// TIA Portal V17 export
// export: Created 2022-02-03T14:45:13.9253235Z, ExportSetting WithDefaults, DisplayName Totally Integrated Automation Portal, DisplayVersion V17, DisplayName TIA Portal Openness, DisplayVersion V17, DisplayName TIA Portal Version Control Interface, DisplayVersion V17, DisplayName SINAMICS Startdrive Advanced, DisplayVersion V17, DisplayName SINAMICS Startdrive G130, G150, S120, S150, SINAMICS MV, S210, DisplayVersion V17, DisplayName SINAMICS Startdrive G110M, G120, G120C, G120D, G120P, G115D, DisplayVersion V17, DisplayName STEP 7 Professional, DisplayVersion V17, DisplayName STEP 7 Safety, DisplayVersion V17, DisplayName WinCC Advanced, DisplayVersion V17
ORGANIZATION_BLOCK "Pull or plug of modules"   // OB83, LAD, PullOrPlugOfModules
VERSION : 0.1
// stored: IsIECCheckEnabled false, SetENOAutomatically false
   VAR_INPUT
      LADDR : HW_IO;   // Hardware identifier
      Event_Class : Byte;   // 16#38/39: module inserted, removed
      Fault_ID : Byte;   // Fault identifier
   END_VAR
   VAR_TEMP
      tempAddress : GEOADDR;
      temp_RetVal : Word;
   END_VAR
   VAR_TEMP   // added for the SCL form of the ladder/FBD networks
      _w1 : Bool;
   END_VAR
BEGIN

REGION Network 1
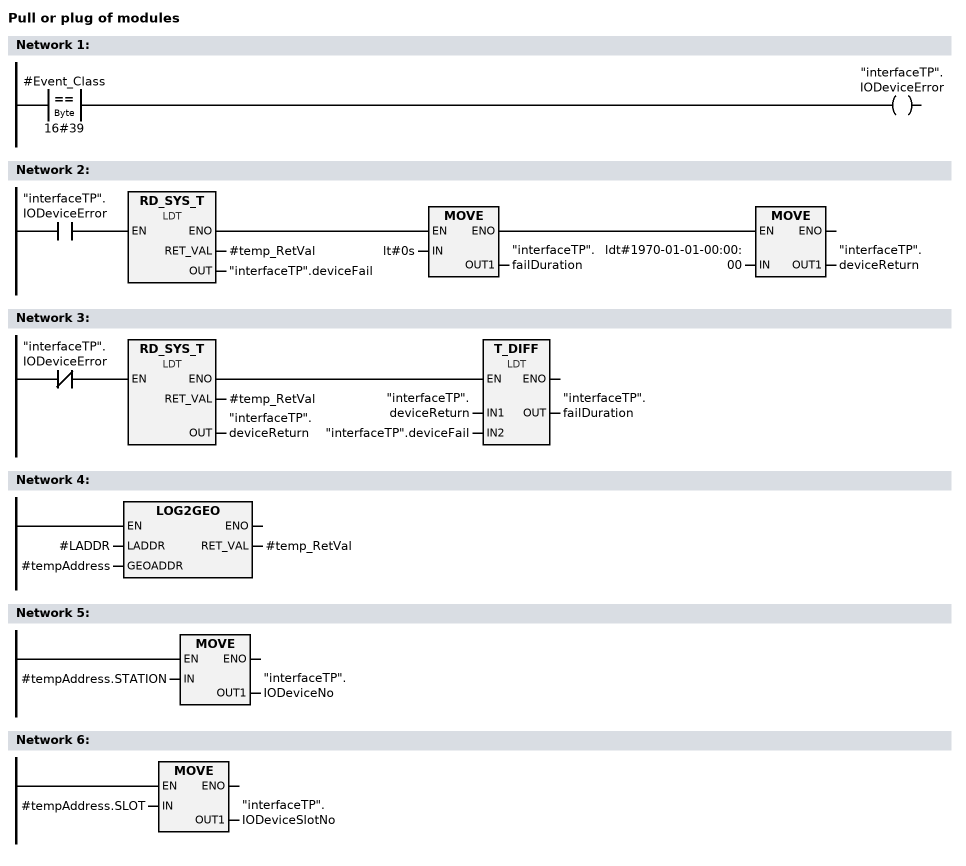
   RUNG wire#powerrail
      { S7_Templates := "SrcType := Byte" } EQ_Contact(in1 := #Event_Class, in2 := 16#39)
      Coil( "interfaceTP".IODeviceError )
   END_RUNG
   // the same network as SCL:
   "interfaceTP".IODeviceError := #Event_Class = 16#39;
END_REGION

REGION Network 2
   RUNG wire#powerrail
      Contact( "interfaceTP".IODeviceError )
      { S7_Templates := "date_type := LDT" } RD_SYS_T(RET_VAL => #temp_RetVal, OUT => "interfaceTP".deviceFail)
      Move(in := lt#0s, out1 => "interfaceTP".failDuration)
      Move(in := ldt#1970-01-01-00:00:00, out1 => "interfaceTP".deviceReturn)
   END_RUNG
   // the same network as SCL:
   #temp_RetVal := RD_SYS_T(EN := "interfaceTP".IODeviceError, OUT => "interfaceTP".deviceFail, ENO => #_w1);
   IF #_w1 THEN
       "interfaceTP".failDuration := lt#0s;
       "interfaceTP".deviceReturn := ldt#1970-01-01-00:00:00;
   END_IF;
END_REGION

REGION Network 3
   RUNG wire#powerrail
      I_Contact( "interfaceTP".IODeviceError )
      { S7_Templates := "date_type := LDT" } RD_SYS_T(RET_VAL => #temp_RetVal, OUT => "interfaceTP".deviceReturn)
      { S7_Templates := "[date_type := LDT, time_type := LTime]" } T_DIFF(IN1 := "interfaceTP".deviceReturn, IN2 := "interfaceTP".deviceFail, OUT => "interfaceTP".failDuration)
   END_RUNG
   // the same network as SCL:
   #temp_RetVal := RD_SYS_T(EN := NOT "interfaceTP".IODeviceError,
                           OUT => "interfaceTP".deviceReturn,
                           ENO => #_w1);
   IF #_w1 THEN
       T_DIFF(IN1 := "interfaceTP".deviceReturn, IN2 := "interfaceTP".deviceFail, OUT => "interfaceTP".failDuration);
   END_IF;
END_REGION

REGION Network 4
   RUNG wire#powerrail
      LOG2GEO(LADDR := #LADDR, GEOADDR := #tempAddress, Ret_Val => #temp_RetVal)
   END_RUNG
   // the same network as SCL:
   #temp_RetVal := LOG2GEO(LADDR := #LADDR, GEOADDR := #tempAddress);
END_REGION

REGION Network 5
   RUNG wire#powerrail
      Move(in := #tempAddress.STATION, out1 => "interfaceTP".IODeviceNo)
   END_RUNG
   // the same network as SCL:
   "interfaceTP".IODeviceNo := #tempAddress.STATION;
END_REGION

REGION Network 6
   RUNG wire#powerrail
      Move(in := #tempAddress.SLOT, out1 => "interfaceTP".IODeviceSlotNo)
   END_RUNG
   // the same network as SCL:
   "interfaceTP".IODeviceSlotNo := #tempAddress.SLOT;
END_REGION
END_ORGANIZATION_BLOCK
